//{attribute 'qualified_only'}
{attribute 'strict'}
TYPE eAuto_State_Macine :
(
	Auto_Stop_State 	:= 0,
	Auto_Init_State 	:= 1,
	Auto_Ready_State 	:= 2,
	Auto_Y_Motion_State := 3,
	Auto_Marking_State 	:= 4
);
END_TYPE

(* stored: Version 1.1.0.1, ProductVersion 3.1.4024.3
   EnumerationTextList eAuto_State_Macine: Id {e45098cb-16f8-49c9-bd2e-7e7db0703c2d} *)
